PROGRAM TEST_AnyBuffer_ReplaceAtIndex
VAR
	// Loop counter
	i						: DINT;
END_VAR

ReplaceAtBeginning();
ReplaceInMiddle();
ReplaceAtEnd();
ReturnsTrueOnSuccess();
ReturnsFalseOnNegativeIndex();
ReturnsFalseOnIndexAtCapacity();
ReturnsFalseOnIndexAboveCapacity();
WrongElementSize();
BufferUnchangedExceptIndex();
MetadataUnchanged();
MultipleReplacements();
ReplaceAllCapacityPositions();
ReplaceWithDifferentValues();
ReplaceSameIndexMultipleTimes();
ReplaceEmptyPosition();
ReplaceWhenBufferEmpty();

// All other elements remain unchanged after replace
METHOD BufferUnchangedExceptIndex
IF TestSuite.Test(__POUNAME()).ExecuteTest() THEN
	// Arrange - [100, 200, 300, 400, 500]
	fbAnyBuffer.Clear();
	FOR i := 1 TO 5 DO
		testElement := i * 100;
		fbAnyBuffer.PushRight(element := testElement);
	END_FOR

	// Act - Replace middle element (index 2)
	testElement := DINT#999;
	Success := fbAnyBuffer.ReplaceAtIndex(index := TEST_LL+2, element := testElement);

	// Assert - Only index 2 should be changed
	TestSuite.Test(__POUNAME()).AssertEqual(TEST_BOOL_TRUE, Success);
	TEST_DINT := 100;
	TestSuite.Test(__POUNAME()).AssertEqual(TEST_DINT, RawBuffer[TEST_LL+0]);
	TEST_DINT := 200;
	TestSuite.Test(__POUNAME()).AssertEqual(TEST_DINT, RawBuffer[TEST_LL+1]);
	TEST_DINT := 999;
	TestSuite.Test(__POUNAME()).AssertEqual(TEST_DINT, RawBuffer[TEST_LL+2]);
	TEST_DINT := 400;
	TestSuite.Test(__POUNAME()).AssertEqual(TEST_DINT, RawBuffer[TEST_LL+3]);
	TEST_DINT := 500;
	TestSuite.Test(__POUNAME()).AssertEqual(TEST_DINT, RawBuffer[TEST_LL+4]);
END_IF
END_METHOD

// ElementCount and all metadata remain unchanged after replace
METHOD MetadataUnchanged
IF TestSuite.Test(__POUNAME()).ExecuteTest() THEN
	// Arrange
	fbAnyBuffer.Clear();
	FOR i := 1 TO TEST_UL-TEST_LL+1 DO
		testElement := i * 100;
		fbAnyBuffer.PushRight(element := testElement);
	END_FOR
	TEST_DINT := 5;
	TestSuite.Test(__POUNAME()).AssertEqual(TEST_DINT, fbAnyBuffer.Metadata.elementCount);
	// Verify capacity was updated by PushRight
	TEST_DINT := 0;
	TestSuite.Test(__POUNAME()).AssertEqual(TEST_DINT, fbAnyBuffer.Metadata.capacity);

	// Act - Replace several elements
	testElement := DINT#111;
	Success := fbAnyBuffer.ReplaceAtIndex(index := TEST_LL, element := testElement);
	TestSuite.Test(__POUNAME()).AssertEqual(TEST_BOOL_TRUE, Success);

	testElement := DINT#333;
	Success := fbAnyBuffer.ReplaceAtIndex(index := TEST_LL+2, element := testElement);
	TestSuite.Test(__POUNAME()).AssertEqual(TEST_BOOL_TRUE, Success);

	testElement := DINT#555;
	Success := fbAnyBuffer.ReplaceAtIndex(index := TEST_LL+4, element := testElement);
	TestSuite.Test(__POUNAME()).AssertEqual(TEST_BOOL_TRUE, Success);

	// Assert - All metadata should be unchanged
	TEST_DINT := 5;
	TestSuite.Test(__POUNAME()).AssertEqual(TEST_DINT, fbAnyBuffer.Metadata.elementCount);
	TEST_DINT := 0;
	TestSuite.Test(__POUNAME()).AssertEqual(TEST_DINT, fbAnyBuffer.Metadata.capacity);
END_IF
END_METHOD

// Sequential replacements at different indices work correctly
METHOD MultipleReplacements
IF TestSuite.Test(__POUNAME()).ExecuteTest() THEN
	// Arrange
	fbAnyBuffer.Clear();
	FOR i := 1 TO TEST_UL-TEST_LL+1 DO
		testElement := i * 100;
		fbAnyBuffer.PushRight(element := testElement);
	END_FOR

	// Act - Replace multiple positions
	testElement := DINT#111;
	Success := fbAnyBuffer.ReplaceAtIndex(index := TEST_LL, element := testElement);
	TestSuite.Test(__POUNAME()).AssertEqual(TEST_BOOL_TRUE, Success);

	testElement := DINT#222;
	Success := fbAnyBuffer.ReplaceAtIndex(index := TEST_LL+1, element := testElement);
	TestSuite.Test(__POUNAME()).AssertEqual(TEST_BOOL_TRUE, Success);

	testElement := DINT#555;
	Success := fbAnyBuffer.ReplaceAtIndex(index := TEST_LL+4, element := testElement);
	TestSuite.Test(__POUNAME()).AssertEqual(TEST_BOOL_TRUE, Success);

	// Assert - All replacements should be successful
	TEST_DINT := 111;
	TestSuite.Test(__POUNAME()).AssertEqual(TEST_DINT, RawBuffer[TEST_LL]);
	TEST_DINT := 222;
	TestSuite.Test(__POUNAME()).AssertEqual(TEST_DINT, RawBuffer[TEST_LL+1]);
	TEST_DINT := 300;
	TestSuite.Test(__POUNAME()).AssertEqual(TEST_DINT, RawBuffer[TEST_LL+2]);
	TEST_DINT := 400;
	TestSuite.Test(__POUNAME()).AssertEqual(TEST_DINT, RawBuffer[TEST_LL+3]);
	TEST_DINT := 555;
	TestSuite.Test(__POUNAME()).AssertEqual(TEST_DINT, RawBuffer[TEST_LL+4]);
END_IF
END_METHOD

// Can replace every capacity position (0 to capacity-1)
METHOD ReplaceAllCapacityPositions
IF TestSuite.Test(__POUNAME()).ExecuteTest() THEN
	// Arrange - Fill buffer completely
	fbAnyBuffer.Clear();
	FOR i := 1 TO TEST_UL-TEST_LL+1 DO
		testElement := i * 100;
		fbAnyBuffer.PushRight(element := testElement);
	END_FOR

	// Act - Replace all capacity positions (0 through capacity-1 = 0 through 4)
	FOR i := TEST_LL TO TEST_UL DO
		testElement := (i-TEST_LL + 1) * 1000;
		Success := fbAnyBuffer.ReplaceAtIndex(index := TO_DINT(i), element := testElement);
		TestSuite.Test(__POUNAME()).AssertEqual(TEST_BOOL_TRUE, Success);
	END_FOR

	// Assert - All positions should be replaced
	TEST_DINT := 1000;
	TestSuite.Test(__POUNAME()).AssertEqual(TEST_DINT, RawBuffer[TEST_LL]);
	TEST_DINT := 2000;
	TestSuite.Test(__POUNAME()).AssertEqual(TEST_DINT, RawBuffer[TEST_LL+1]);
	TEST_DINT := 3000;
	TestSuite.Test(__POUNAME()).AssertEqual(TEST_DINT, RawBuffer[TEST_LL+2]);
	TEST_DINT := 4000;
	TestSuite.Test(__POUNAME()).AssertEqual(TEST_DINT, RawBuffer[TEST_LL+3]);
	TEST_DINT := 5000;
	TestSuite.Test(__POUNAME()).AssertEqual(TEST_DINT, RawBuffer[TEST_LL+4]);
	// Metadata unchanged
	TEST_DINT := 5;
	TestSuite.Test(__POUNAME()).AssertEqual(TEST_DINT, fbAnyBuffer.Metadata.elementCount);
END_IF
END_METHOD

// Replacing at index 0 updates first element correctly
METHOD ReplaceAtBeginning
IF TestSuite.Test(__POUNAME()).ExecuteTest() THEN
	// Arrange
	fbAnyBuffer.Clear();
	testElement := DINT#100;
	fbAnyBuffer.PushRight(element := testElement);
	testElement := DINT#200;
	fbAnyBuffer.PushRight(element := testElement);
	testElement := DINT#300;
	fbAnyBuffer.PushRight(element := testElement);

	// Act - Replace first element
	testElement := DINT#999;
	Success := fbAnyBuffer.ReplaceAtIndex(index := TEST_LL, element := testElement);

	// Assert
	TestSuite.Test(__POUNAME()).AssertEqual(TEST_BOOL_TRUE, Success);
	TEST_DINT := 999;
	TestSuite.Test(__POUNAME()).AssertEqual(TEST_DINT, RawBuffer[TEST_LL]);
	TEST_DINT := 200;
	TestSuite.Test(__POUNAME()).AssertEqual(TEST_DINT, RawBuffer[TEST_LL+1]);
	TEST_DINT := 300;
	TestSuite.Test(__POUNAME()).AssertEqual(TEST_DINT, RawBuffer[TEST_LL+2]);
	TEST_DINT := 3;
	TestSuite.Test(__POUNAME()).AssertEqual(TEST_DINT, fbAnyBuffer.Metadata.elementCount);
END_IF
END_METHOD

// Replacing at last capacity index updates last element
METHOD ReplaceAtEnd
IF TestSuite.Test(__POUNAME()).ExecuteTest() THEN
	// Arrange - fill buffer to capacity
	fbAnyBuffer.Clear();
	testElement := DINT#100;
	fbAnyBuffer.PushRight(element := testElement);
	testElement := DINT#200;
	fbAnyBuffer.PushRight(element := testElement);
	testElement := DINT#300;
	fbAnyBuffer.PushRight(element := testElement);
	testElement := DINT#400;
	fbAnyBuffer.PushRight(element := testElement);
	testElement := DINT#500;
	fbAnyBuffer.PushRight(element := testElement);

	// Act - Replace last capacity position (index 4 = capacity-1)
	testElement := DINT#999;
	Success := fbAnyBuffer.ReplaceAtIndex(index := TEST_LL+4, element := testElement);

	// Assert
	TestSuite.Test(__POUNAME()).AssertEqual(TEST_BOOL_TRUE, Success);
	TEST_DINT := 100;
	TestSuite.Test(__POUNAME()).AssertEqual(TEST_DINT, RawBuffer[TEST_LL]);
	TEST_DINT := 200;
	TestSuite.Test(__POUNAME()).AssertEqual(TEST_DINT, RawBuffer[TEST_LL+1]);
	TEST_DINT := 300;
	TestSuite.Test(__POUNAME()).AssertEqual(TEST_DINT, RawBuffer[TEST_LL+2]);
	TEST_DINT := 400;
	TestSuite.Test(__POUNAME()).AssertEqual(TEST_DINT, RawBuffer[TEST_LL+3]);
	TEST_DINT := 999;
	TestSuite.Test(__POUNAME()).AssertEqual(TEST_DINT, RawBuffer[TEST_LL+4]);
	// Metadata unchanged
	TEST_DINT := 5;
	TestSuite.Test(__POUNAME()).AssertEqual(TEST_DINT, fbAnyBuffer.Metadata.elementCount);
END_IF
END_METHOD

// Can replace position that was never filled (elementCount < index < capacity)
METHOD ReplaceEmptyPosition
IF TestSuite.Test(__POUNAME()).ExecuteTest() THEN
	// Arrange - only fill first 2 positions
	fbAnyBuffer.Clear();
	testElement := DINT#100;
	fbAnyBuffer.PushRight(element := testElement);
	testElement := DINT#200;
	fbAnyBuffer.PushRight(element := testElement);
	// elementCount = 2, but capacity = 5, so indices 2, 3, 4 are "empty"

	// Act - Replace position 3 (which was never logically filled)
	testElement := DINT#999;
	Success := fbAnyBuffer.ReplaceAtIndex(index := TEST_LL+3, element := testElement);

	// Assert - Should succeed because index 3 is within capacity
	TestSuite.Test(__POUNAME()).AssertEqual(TEST_BOOL_TRUE, Success);
	TEST_DINT := 999;
	TestSuite.Test(__POUNAME()).AssertEqual(TEST_DINT, RawBuffer[TEST_LL+3]);

	// Metadata should remain unchanged
	TEST_DINT := 2;
	TestSuite.Test(__POUNAME()).AssertEqual(TEST_DINT, fbAnyBuffer.Metadata.elementCount);
END_IF
END_METHOD

// Replacing at middle index updates correct element
METHOD ReplaceInMiddle
IF TestSuite.Test(__POUNAME()).ExecuteTest() THEN
	// Arrange
	fbAnyBuffer.Clear();
	testElement := DINT#100;
	fbAnyBuffer.PushRight(element := testElement);
	testElement := DINT#200;
	fbAnyBuffer.PushRight(element := testElement);
	testElement := DINT#300;
	fbAnyBuffer.PushRight(element := testElement);
	testElement := DINT#400;
	fbAnyBuffer.PushRight(element := testElement);

	// Act - Replace middle element (index 1)
	testElement := DINT#999;
	Success := fbAnyBuffer.ReplaceAtIndex(index := TEST_LL+1, element := testElement);

	// Assert
	TestSuite.Test(__POUNAME()).AssertEqual(TEST_BOOL_TRUE, Success);
	TEST_DINT := 100;
	TestSuite.Test(__POUNAME()).AssertEqual(TEST_DINT, RawBuffer[TEST_LL+0]);
	TEST_DINT := 999;
	TestSuite.Test(__POUNAME()).AssertEqual(TEST_DINT, RawBuffer[TEST_LL+1]);
	TEST_DINT := 300;
	TestSuite.Test(__POUNAME()).AssertEqual(TEST_DINT, RawBuffer[TEST_LL+2]);
	TEST_DINT := 400;
	TestSuite.Test(__POUNAME()).AssertEqual(TEST_DINT, RawBuffer[TEST_LL+3]);
	TEST_DINT := 4;
	TestSuite.Test(__POUNAME()).AssertEqual(TEST_DINT, fbAnyBuffer.Metadata.elementCount);
END_IF
END_METHOD

// Can overwrite same position repeatedly
METHOD ReplaceSameIndexMultipleTimes
IF TestSuite.Test(__POUNAME()).ExecuteTest() THEN
	// Arrange
	fbAnyBuffer.Clear();
	testElement := DINT#100;
	fbAnyBuffer.PushRight(element := testElement);
	testElement := DINT#200;
	fbAnyBuffer.PushRight(element := testElement);
	testElement := DINT#300;
	fbAnyBuffer.PushRight(element := testElement);

	// Act - Replace same index multiple times
	testElement := DINT#111;
	Success := fbAnyBuffer.ReplaceAtIndex(index := TEST_LL+1, element := testElement);
	TestSuite.Test(__POUNAME()).AssertEqual(TEST_BOOL_TRUE, Success);
	TEST_DINT := 111;
	TestSuite.Test(__POUNAME()).AssertEqual(TEST_DINT, RawBuffer[TEST_LL+1]);

	testElement := DINT#222;
	Success := fbAnyBuffer.ReplaceAtIndex(index := TEST_LL+1, element := testElement);
	TestSuite.Test(__POUNAME()).AssertEqual(TEST_BOOL_TRUE, Success);
	TEST_DINT := 222;
	TestSuite.Test(__POUNAME()).AssertEqual(TEST_DINT, RawBuffer[TEST_LL+1]);

	testElement := DINT#333;
	Success := fbAnyBuffer.ReplaceAtIndex(index := TEST_LL+1, element := testElement);
	TestSuite.Test(__POUNAME()).AssertEqual(TEST_BOOL_TRUE, Success);
	TEST_DINT := 333;
	TestSuite.Test(__POUNAME()).AssertEqual(TEST_DINT, RawBuffer[TEST_LL+1]);

	// Assert - Other elements unchanged, count unchanged
	TEST_DINT := 100;
	TestSuite.Test(__POUNAME()).AssertEqual(TEST_DINT, RawBuffer[TEST_LL+0]);
	TEST_DINT := 300;
	TestSuite.Test(__POUNAME()).AssertEqual(TEST_DINT, RawBuffer[TEST_LL+2]);
	TEST_DINT := 3;
	TestSuite.Test(__POUNAME()).AssertEqual(TEST_DINT, fbAnyBuffer.Metadata.elementCount);
END_IF
END_METHOD

// Replace succeeds even when elementCount = 0 (if index < capacity)
METHOD ReplaceWhenBufferEmpty
IF TestSuite.Test(__POUNAME()).ExecuteTest() THEN
	// Arrange - empty buffer (elementCount = 0)
	fbAnyBuffer.Clear();
	// Buffer is empty, but capacity is 5, so indices 0-4 are valid

	// Act - Replace at various positions in empty buffer
	testElement := DINT#111;
	Success := fbAnyBuffer.ReplaceAtIndex(index := TEST_LL, element := testElement);
	TestSuite.Test(__POUNAME()).AssertEqual(TEST_BOOL_TRUE, Success);
	TEST_DINT := 111;
	TestSuite.Test(__POUNAME()).AssertEqual(TEST_DINT, RawBuffer[TEST_LL]);

	testElement := DINT#333;
	Success := fbAnyBuffer.ReplaceAtIndex(index := TEST_LL+2, element := testElement);
	TestSuite.Test(__POUNAME()).AssertEqual(TEST_BOOL_TRUE, Success);
	TEST_DINT := 333;
	TestSuite.Test(__POUNAME()).AssertEqual(TEST_DINT, RawBuffer[TEST_LL+2]);

	testElement := DINT#555;
	Success := fbAnyBuffer.ReplaceAtIndex(index := TEST_LL+4, element := testElement);
	TestSuite.Test(__POUNAME()).AssertEqual(TEST_BOOL_TRUE, Success);
	TEST_DINT := 555;
	TestSuite.Test(__POUNAME()).AssertEqual(TEST_DINT, RawBuffer[TEST_LL+4]);

	// Metadata should remain unchanged (still empty from logical perspective)
	TEST_DINT := 0;
	TestSuite.Test(__POUNAME()).AssertEqual(TEST_DINT, fbAnyBuffer.Metadata.elementCount);
END_IF
END_METHOD

// Replace works with various data values
METHOD ReplaceWithDifferentValues
IF TestSuite.Test(__POUNAME()).ExecuteTest() THEN
	// Arrange
	fbAnyBuffer.Clear();
	FOR i := TEST_LL-TEST_LL+1  TO TEST_UL-TEST_LL+1 DO
		testElement := i * 100;
		fbAnyBuffer.PushRight(element := testElement);
	END_FOR

	// Act - Replace with various values (zero, negative, large)
	testElement := DINT#0;
	Success := fbAnyBuffer.ReplaceAtIndex(index := TEST_LL+0, element := testElement);
	TestSuite.Test(__POUNAME()).AssertEqual(TEST_BOOL_TRUE, Success);

	testElement := DINT#-999;
	Success := fbAnyBuffer.ReplaceAtIndex(index := TEST_LL+2, element := testElement);
	TestSuite.Test(__POUNAME()).AssertEqual(TEST_BOOL_TRUE, Success);

	testElement := DINT#2147483647;  // Max DINT
	Success := fbAnyBuffer.ReplaceAtIndex(index := TEST_LL+4, element := testElement);
	TestSuite.Test(__POUNAME()).AssertEqual(TEST_BOOL_TRUE, Success);

	// Assert - All values replaced correctly
	TEST_DINT := 0;
	TestSuite.Test(__POUNAME()).AssertEqual(TEST_DINT, RawBuffer[TEST_LL+0]);
	TEST_DINT := 200;
	TestSuite.Test(__POUNAME()).AssertEqual(TEST_DINT, RawBuffer[TEST_LL+1]);
	TEST_DINT := -999;
	TestSuite.Test(__POUNAME()).AssertEqual(TEST_DINT, RawBuffer[TEST_LL+2]);
	TEST_DINT := 400;
	TestSuite.Test(__POUNAME()).AssertEqual(TEST_DINT, RawBuffer[TEST_LL+3]);
	TEST_DINT := 2147483647;
	TestSuite.Test(__POUNAME()).AssertEqual(TEST_DINT, RawBuffer[TEST_LL+4]);
END_IF
END_METHOD

// FALSE returned when index > capacity
METHOD ReturnsFalseOnIndexAboveCapacity
IF TestSuite.Test(__POUNAME()).ExecuteTest() THEN
	// Arrange - capacity is 5
	fbAnyBuffer.Clear();
	testElement := DINT#100;
	fbAnyBuffer.PushRight(element := testElement);
	testElement := DINT#200;
	fbAnyBuffer.PushRight(element := testElement);

	// Act & Assert - Try index much larger than capacity
	testElement := DINT#999;
	Success := fbAnyBuffer.ReplaceAtIndex(index := TEST_UL+100, element := testElement);
	TestSuite.Test(__POUNAME()).AssertEqual(TEST_BOOL_FALSE, Success);

	// Act & Assert - Try another large index
	Success := fbAnyBuffer.ReplaceAtIndex(index := TEST_UL+10, element := testElement);
	TestSuite.Test(__POUNAME()).AssertEqual(TEST_BOOL_FALSE, Success);
END_IF
END_METHOD

// FALSE returned when index == capacity
METHOD ReturnsFalseOnIndexAtCapacity
IF TestSuite.Test(__POUNAME()).ExecuteTest() THEN
	// Arrange - capacity is 5
	fbAnyBuffer.Clear();
	testElement := DINT#100;
	fbAnyBuffer.PushRight(element := testElement);

	// Act - Try to replace beyond last index
	testElement := DINT#999;
	Success := fbAnyBuffer.ReplaceAtIndex(index := TEST_LL+5, element := testElement);

	// Assert
	TestSuite.Test(__POUNAME()).AssertEqual(TEST_BOOL_FALSE, Success);
END_IF
END_METHOD

// FALSE returned for negative index
METHOD ReturnsFalseOnNegativeIndex
IF TestSuite.Test(__POUNAME()).ExecuteTest() THEN
	// Arrange
	fbAnyBuffer.Clear();
	testElement := DINT#100;
	fbAnyBuffer.PushRight(element := testElement);

	// Act
	testElement := DINT#999;
	Success := fbAnyBuffer.ReplaceAtIndex(index := TEST_LL-1, element := testElement);

	// Assert
	TestSuite.Test(__POUNAME()).AssertEqual(TEST_BOOL_FALSE, Success);
	TEST_DINT := 1;
	TestSuite.Test(__POUNAME()).AssertEqual(TEST_DINT, fbAnyBuffer.Metadata.elementCount);
	TEST_DINT := 100;
	TestSuite.Test(__POUNAME()).AssertEqual(TEST_DINT, RawBuffer[TEST_LL+0]);
END_IF
END_METHOD

// Method returns TRUE when replace succeeds
METHOD ReturnsTrueOnSuccess
IF TestSuite.Test(__POUNAME()).ExecuteTest() THEN
	// Arrange
	fbAnyBuffer.Clear();
	testElement := DINT#100;
	fbAnyBuffer.PushRight(element := testElement);
	testElement := DINT#200;
	fbAnyBuffer.PushRight(element := testElement);

	// Act
	testElement := DINT#999;
	Success := fbAnyBuffer.ReplaceAtIndex(index := TEST_LL, element := testElement);

	// Assert
	TestSuite.Test(__POUNAME()).AssertEqual(TEST_BOOL_TRUE, Success);
END_IF
END_METHOD

// FALSE returned when element size doesn't match
METHOD WrongElementSize
IF TestSuite.Test(__POUNAME()).ExecuteTest() THEN
	// Arrange
	fbAnyBuffer.Clear();
	testElement := DINT#100;
	fbAnyBuffer.PushRight(element := testElement);

	// Act - Try to replace with wrong element size
	Success := fbAnyBuffer.ReplaceAtIndex(index := TEST_LL, element := WrongSizeElement);

	// Assert - Should fail (IN and DINT are different size)
	TestSuite.Test(__POUNAME()).AssertEqual(TEST_BOOL_FALSE, Success);

	// Verify buffer element count unchanged
	TEST_DINT := 1;
	TestSuite.Test(__POUNAME()).AssertEqual(TEST_DINT, fbAnyBuffer.Metadata.elementCount);
END_IF
END_METHOD

END_PROGRAM

(* stored: Version 1.1.0.1, ProductVersion 3.1.4026.18
   POU TEST_AnyBuffer_ReplaceAtIndex: Id {d5e6f7a8-9012-34ef-ab67-890123def456}, SpecialFunc None
   Method BufferUnchangedExceptIndex: Id {11223344-5566-7788-99aa-bbccddee1122}
   Method MetadataUnchanged: Id {22334455-6677-8899-aabb-ccddeeaa2233}
   Method MultipleReplacements: Id {33445566-7788-99aa-bbcc-ddeeff003344}
   Method ReplaceAllCapacityPositions: Id {44556677-8899-aabb-ccdd-eeff00444455}
   Method ReplaceAtBeginning: Id {55667788-99aa-bbcc-ddee-ff0011225566}
   Method ReplaceAtEnd: Id {66778899-aabb-ccdd-eeff-001122336677}
   Method ReplaceEmptyPosition: Id {50f1f761-3d82-446f-943f-fdd0c0d24206}
   Method ReplaceInMiddle: Id {778899aa-bbcc-ddee-ff00-112233447788}
   Method ReplaceSameIndexMultipleTimes: Id {8899aabb-ccdd-eeff-0011-223344558899}
   Method ReplaceWhenBufferEmpty: Id {f48a97da-a4b4-4112-a4e5-0ae6ab1afb48}
   Method ReplaceWithDifferentValues: Id {99aabbcc-ddee-ff00-1122-3344556699aa}
   Method ReturnsFalseOnIndexAboveCapacity: Id {bbccddee-ff00-1122-3344-5566bbccddee}
   Method ReturnsFalseOnIndexAtCapacity: Id {aabbccdd-eeff-0011-2233-445566aabbcc}
   Method ReturnsFalseOnNegativeIndex: Id {ccddeeff-0011-2233-4455-66ccddeeff00}
   Method ReturnsTrueOnSuccess: Id {ddeeff00-1122-3344-5566-77ddeeff0011}
   Method WrongElementSize: Id {eeff0011-2233-4455-6677-88eeff001122} *)
